FUNCTION_BLOCK Emitr
  (* Standard: 61499-2 *)
  (* Compiler header: Emitr.h *)
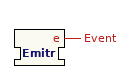
  EVENT_OUTPUT
    e;
  END_EVENT
END_FUNCTION_BLOCK
